INTERFACE I_Command EXTENDS __SYSTEM.IQueryInterface

{attribute 'monitoring' := 'call'}
PROPERTY Description : STRING
GET
END_GET
END_PROPERTY

METHOD Execute : E_Progress
VAR_INPUT
END_VAR
END_METHOD

END_INTERFACE

(* stored: Version 1.1.0.1
   Itf I_Command: Id {6ac1caa1-9aa1-46a4-a975-a161e8b4cef4}
   Property Description: Id {c5cf10c0-d473-4e4f-a074-c70e9881658d}
   Get Get: Id {ceaab77b-fce3-4f05-8452-3596b29a365b}
   Method Execute: Id {a051ecf4-eb8f-4ded-b2a2-38f5d78bc77e} *)
